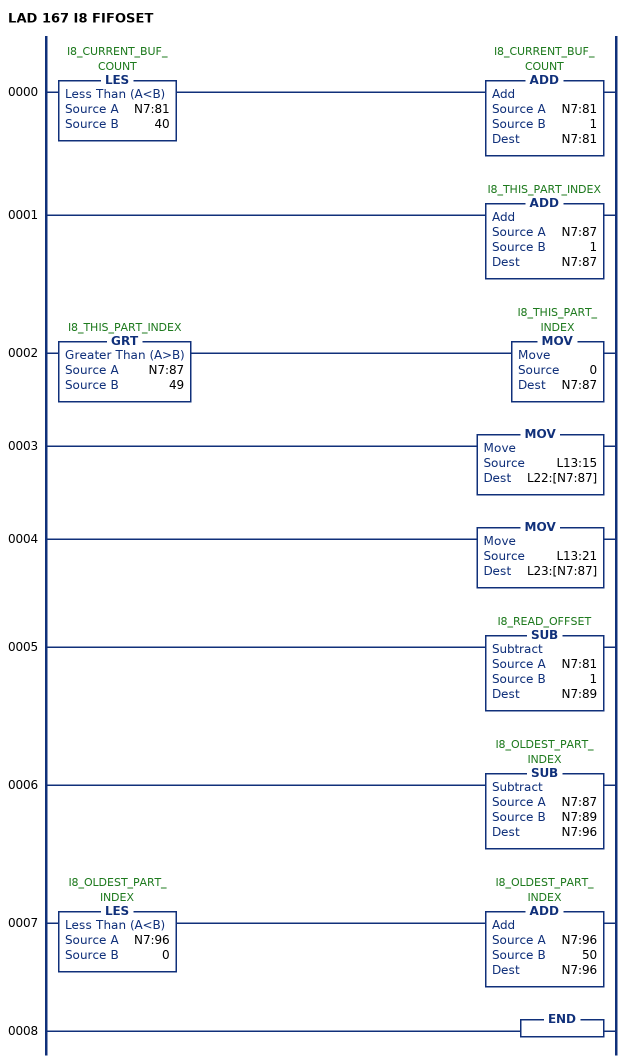
% Rung: 0 %
SOR LES N7:81 40 ADD N7:81 1 N7:81 EOR
%   N7:81  I8_CURRENT_BUF_COUNT %
% Rung: 1 %
SOR ADD N7:87 1 N7:87 EOR
%   N7:87  I8_THIS_PART_INDEX %
% Rung: 2 %
SOR GRT N7:87 49 MOV 0 N7:87 EOR
%   N7:87  I8_THIS_PART_INDEX %
% Rung: 3 %
SOR MOV L13:15 L22:[N7:87] EOR
%   L13:15  THE_TIME %
%   N7:87  I8_THIS_PART_INDEX %
% Rung: 4 %
SOR MOV L13:21 L23:[N7:87] EOR
%   L13:21  TOP_POSITION %
%   N7:87  I8_THIS_PART_INDEX %
% Rung: 5 %
SOR SUB N7:81 1 N7:89 EOR
%   N7:81  I8_CURRENT_BUF_COUNT %
%   N7:89  I8_READ_OFFSET %
% Rung: 6 %
SOR SUB N7:87 N7:89 N7:96 EOR
%   N7:87  I8_THIS_PART_INDEX %
%   N7:89  I8_READ_OFFSET %
%   N7:96  I8_OLDEST_PART_INDEX %
% Rung: 7 %
SOR LES N7:96 0 ADD N7:96 50 N7:96 EOR
%   N7:96  I8_OLDEST_PART_INDEX %
% Rung: 8 %
SOR END EOR

LADDER 168 "I8 FIFOGET"
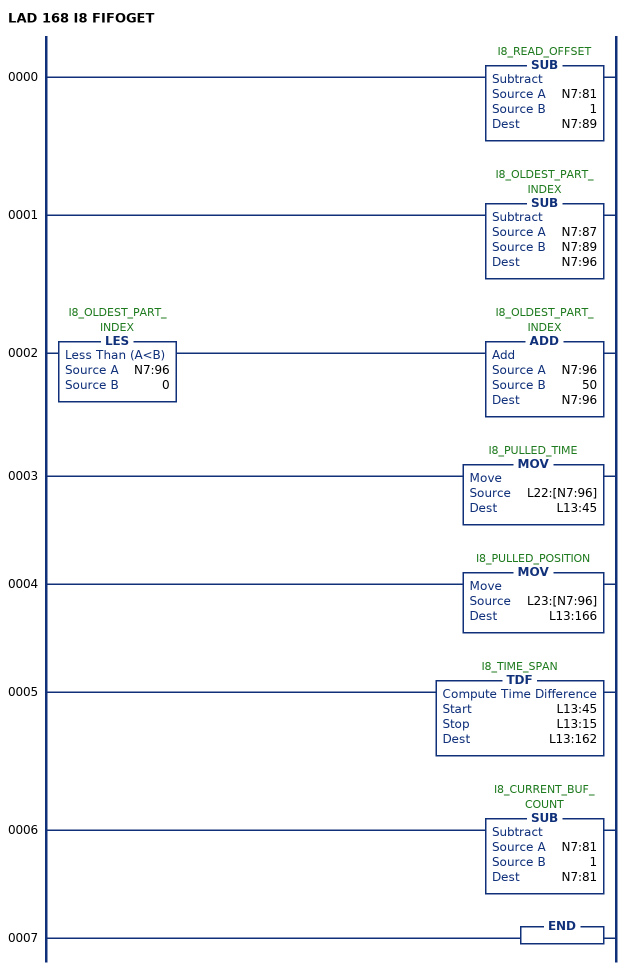
% Rung: 0 %
SOR SUB N7:81 1 N7:89 EOR
%   N7:81  I8_CURRENT_BUF_COUNT %
%   N7:89  I8_READ_OFFSET %
% Rung: 1 %
SOR SUB N7:87 N7:89 N7:96 EOR
%   N7:87  I8_THIS_PART_INDEX %
%   N7:89  I8_READ_OFFSET %
%   N7:96  I8_OLDEST_PART_INDEX %
% Rung: 2 %
SOR LES N7:96 0 ADD N7:96 50 N7:96 EOR
%   N7:96  I8_OLDEST_PART_INDEX %
% Rung: 3 %
SOR MOV L22:[N7:96] L13:45 EOR
%   N7:96  I8_OLDEST_PART_INDEX %
%   L13:45  I8_PULLED_TIME %
% Rung: 4 %
SOR MOV L23:[N7:96] L13:166 EOR
%   N7:96  I8_OLDEST_PART_INDEX %
%   L13:166  I8_PULLED_POSITION %
% Rung: 5 %
SOR TDF L13:45 L13:15 L13:162 EOR
%   L13:45  I8_PULLED_TIME %
%   L13:15  THE_TIME %
%   L13:162  I8_TIME_SPAN %
% Rung: 6 %
SOR SUB N7:81 1 N7:81 EOR
%   N7:81  I8_CURRENT_BUF_COUNT %
% Rung: 7 %
SOR END EOR

LADDER 169 "I8 DATA"
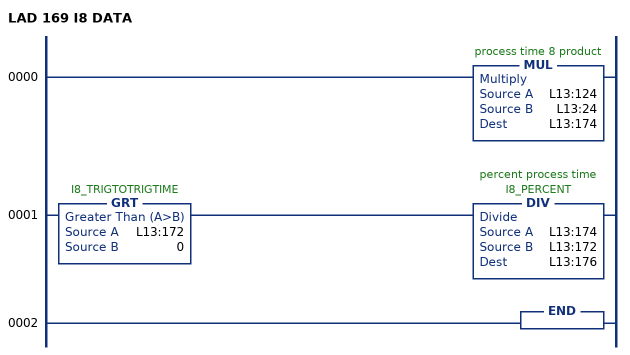
% Rung: 0 %
SOR MUL L13:124 L13:24 L13:174 EOR
%   L13:124  I8_PROCESSTIME %
%   L13:24  "multiplyer to make devision come out to a percentage" %
%   L13:174  "process time 8 product" %
% Rung: 1 %
SOR GRT L13:172 0 DIV L13:174 L13:172 L13:176 EOR
%   L13:172  I8_TRIGTOTRIGTIME %
%   L13:174  "process time 8 product" %
%   L13:176  I8_PERCENT  "percent process time" %
% Rung: 2 %
SOR END EOR

LADDER 170 "I8 FAULT"
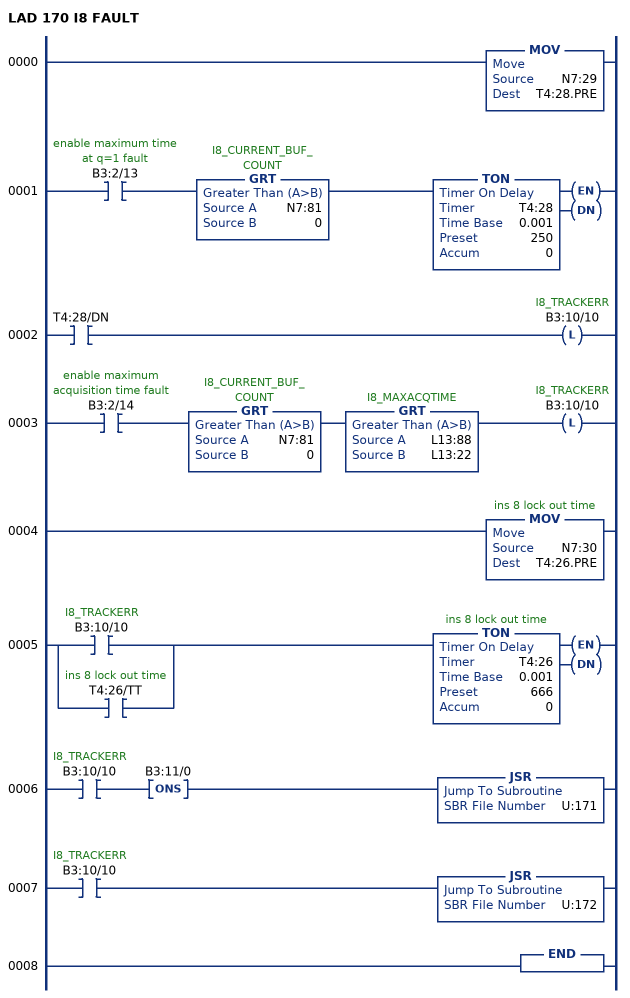
% Rung: 0 %
SOR MOV N7:29 T4:28.PRE EOR
%   N7:29  "max allowed ms time for q to be above 1 if safe fault is used" %
% Rung: 1 %
SOR XIC B3:2/13 GRT N7:81 0 TON T4:28 0.001 250 0 EOR
%   B3:2/13  "enable maximum time at q=1 fault" %
%   N7:81  I8_CURRENT_BUF_COUNT %
% Rung: 2 %
SOR XIC T4:28/DN OTL B3:10/10 EOR
%   B3:10/10  I8_TRACKERR %
% Rung: 3 %
SOR XIC B3:2/14 GRT N7:81 0 GRT L13:88 L13:22 OTL B3:10/10 EOR
%   B3:2/14  "enable maximum acquisition time fault" %
%   N7:81  I8_CURRENT_BUF_COUNT %
%   L13:88  I8_MAXACQTIME %
%   L13:22  "maximum of the longest acquire time allowed if maximum acquire time fault is enabled" %
%   B3:10/10  I8_TRACKERR %
% Rung: 4 %
SOR MOV N7:30 T4:26.PRE EOR
%   N7:30  "ms time setting to lock out inspection to give all pending images a chance to clear" %
%   T4:26  "ins 8 lock out time" %
% Rung: 5 %
SOR BST XIC B3:10/10 NXB XIC T4:26/TT BND TON T4:26 0.001 666 0 EOR
%   B3:10/10  I8_TRACKERR %
%   T4:26  "ins 8 lock out time" %
% Rung: 6 %
SOR XIC B3:10/10 ONS B3:11/0 JSR U:171 EOR
%   B3:10/10  I8_TRACKERR %
% Rung: 7 %
SOR XIC B3:10/10 JSR U:172 EOR
%   B3:10/10  I8_TRACKERR %
% Rung: 8 %
SOR END EOR

LADDER 171 "I8 FIX1"
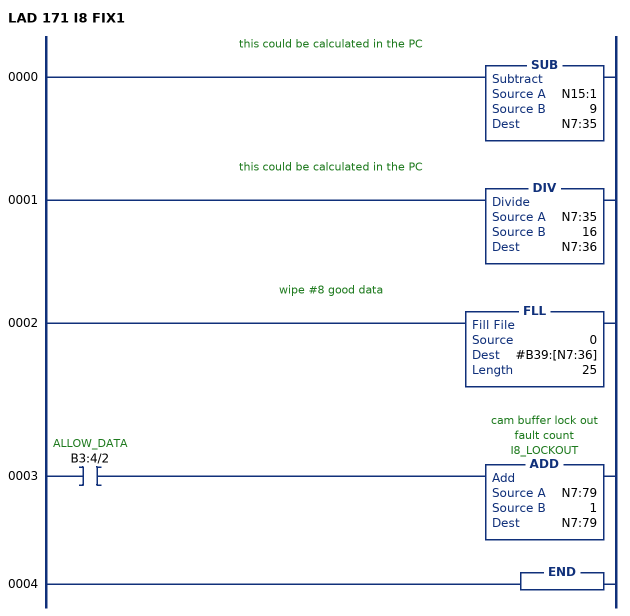
% Rung: 0 %
% this could be calculated in the PC %
SOR SUB N15:1 9 N7:35 EOR
%   N15:1  I8_TRIG_LOC %
% Rung: 1 %
% this could be calculated in the PC %
SOR DIV N7:35 16 N7:36 EOR
% Rung: 2 %
% wipe #8 good data %
SOR FLL 0 #B39:[N7:36] 25 EOR
% Rung: 3 %
SOR XIC B3:4/2 ADD N7:79 1 N7:79 EOR
%   B3:4/2  ALLOW_DATA %
%   N7:79  I8_LOCKOUT  "cam buffer lock out fault count" %
% Rung: 4 %
SOR END EOR

LADDER 172 "I8 FIX2"
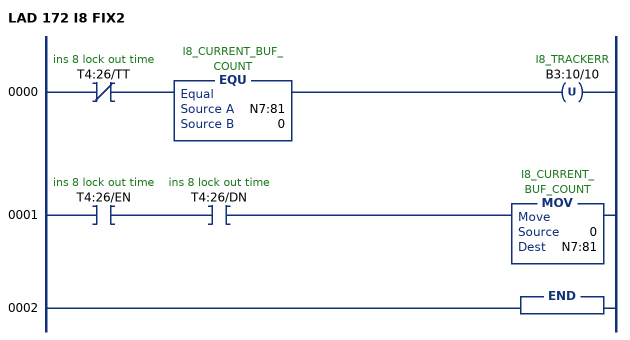
% Rung: 0 %
SOR XIO T4:26/TT EQU N7:81 0 OTU B3:10/10 EOR
%   T4:26  "ins 8 lock out time" %
%   N7:81  I8_CURRENT_BUF_COUNT %
%   B3:10/10  I8_TRACKERR %
% Rung: 1 %
SOR XIC T4:26/EN XIC T4:26/DN MOV 0 N7:81 EOR
%   T4:26  "ins 8 lock out time" %
%   N7:81  I8_CURRENT_BUF_COUNT %
% Rung: 2 %
SOR END EOR

LADDER 200 "PASS BLOW"
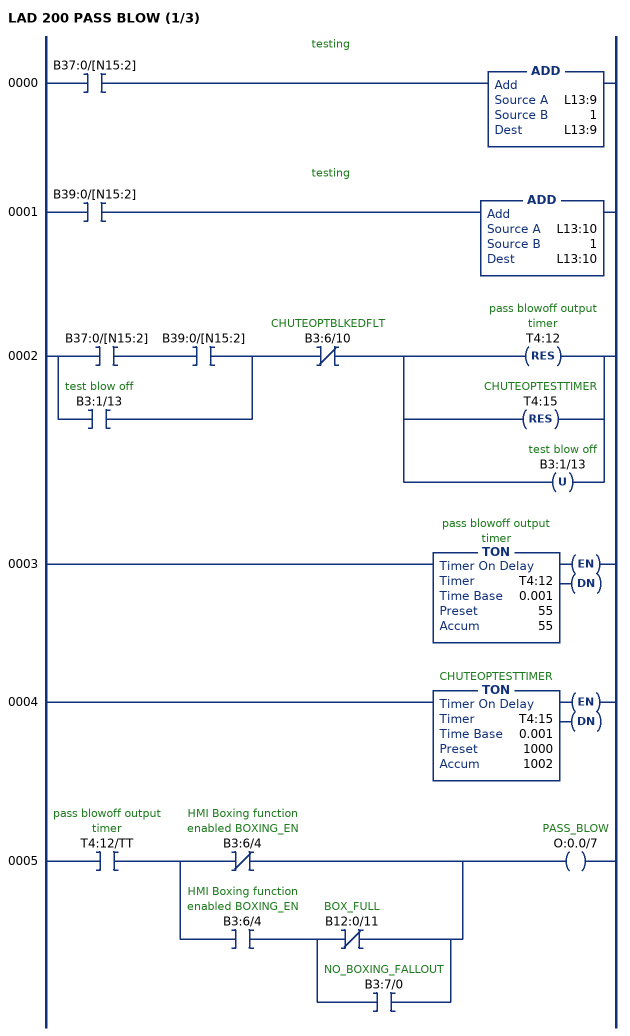
% Rung: 0 %
% testing %
SOR XIC B37:0/[N15:2] ADD L13:9 1 L13:9 EOR
%   B37:0  TOPGOOD1 %
%   N15:2  BLOW_PT %
% Rung: 1 %
% testing %
SOR XIC B39:0/[N15:2] ADD L13:10 1 L13:10 EOR
%   B39:0  TOPGOOD2 %
%   N15:2  BLOW_PT %
% Rung: 2 %
SOR BST XIC B37:0/[N15:2] XIC B39:0/[N15:2] NXB XIC B3:1/13 BND XIO B3:6/10 BST RES T4:12 NXB RES T4:15 NXB OTU B3:1/13 BND EOR
%   B37:0  TOPGOOD1 %
%   N15:2  BLOW_PT %
%   B39:0  TOPGOOD2 %
%   B3:1/13  "test blow off" %
%   B3:6/10  CHUTEOPTBLKEDFLT %
%   T4:12  "pass blowoff output timer" %
%   T4:15  CHUTEOPTESTTIMER %
% Rung: 3 %
SOR TON T4:12 0.001 55 55 EOR
%   T4:12  "pass blowoff output timer" %
% Rung: 4 %
SOR TON T4:15 0.001 1000 1002 EOR
%   T4:15  CHUTEOPTESTTIMER %
% Rung: 5 %
SOR XIC T4:12/TT BST XIO B3:6/4 NXB XIC B3:6/4 BST XIO B12:0/11 NXB XIC B3:7/0 BND BND OTE O:0.0/7 EOR
%   T4:12  "pass blowoff output timer" %
%   B3:6/4  BOXING_EN  "HMI Boxing function enabled" %
%   B12:0/11  BOX_FULL %
%   B3:7/0  NO_BOXING_FALLOUT %
%   O:0.0/7  PASS_BLOW %

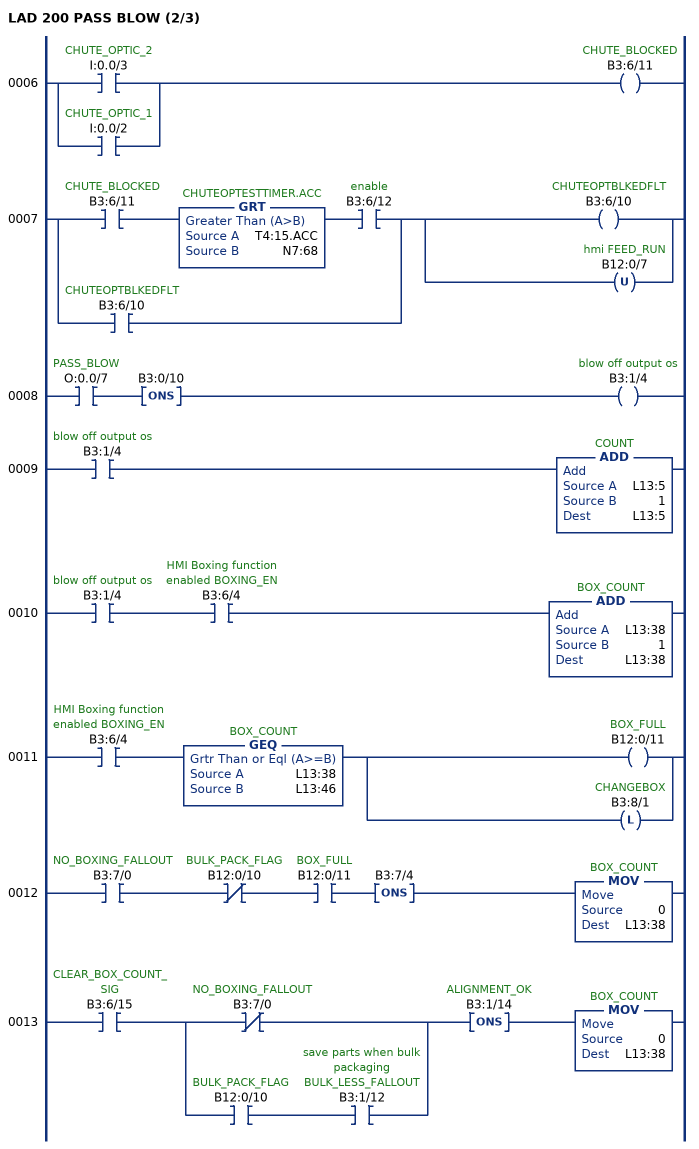
% Rung: 6 %
SOR BST XIC I:0.0/3 NXB XIC I:0.0/2 BND OTE B3:6/11 EOR
%   I:0.0/3  CHUTE_OPTIC_2 %
%   I:0.0/2  CHUTE_OPTIC_1 %
%   B3:6/11  CHUTE_BLOCKED %
% Rung: 7 %
SOR BST XIC B3:6/11 GRT T4:15.ACC N7:68 XIC B3:6/12 NXB XIC B3:6/10 BND BST OTE B3:6/10 NXB OTU B12:0/7 BND EOR
%   B3:6/11  CHUTE_BLOCKED %
%   T4:15  CHUTEOPTESTTIMER %
%   B3:6/12  "enable" %
%   B3:6/10  CHUTEOPTBLKEDFLT %
%   B12:0/7  FEED_RUN  "hmi" %
% Rung: 8 %
SOR XIC O:0.0/7 ONS B3:0/10 OTE B3:1/4 EOR
%   O:0.0/7  PASS_BLOW %
%   B3:1/4  "blow off output os" %
% Rung: 9 %
SOR XIC B3:1/4 ADD L13:5 1 L13:5 EOR
%   B3:1/4  "blow off output os" %
%   L13:5  COUNT %
% Rung: 10 %
SOR XIC B3:1/4 XIC B3:6/4 ADD L13:38 1 L13:38 EOR
%   B3:1/4  "blow off output os" %
%   B3:6/4  BOXING_EN  "HMI Boxing function enabled" %
%   L13:38  BOX_COUNT %
% Rung: 11 %
SOR XIC B3:6/4 GEQ L13:38 L13:46 BST OTE B12:0/11 NXB OTL B3:8/1 BND EOR
%   B3:6/4  BOXING_EN  "HMI Boxing function enabled" %
%   L13:38  BOX_COUNT %
%   L13:46  BOX_LIMIT  "box count setpoint" %
%   B12:0/11  BOX_FULL %
%   B3:8/1  CHANGEBOX %
% Rung: 12 %
SOR XIC B3:7/0 XIO B12:0/10 XIC B12:0/11 ONS B3:7/4 MOV 0 L13:38 EOR
%   B3:7/0  NO_BOXING_FALLOUT %
%   B12:0/10  BULK_PACK_FLAG %
%   B12:0/11  BOX_FULL %
%   L13:38  BOX_COUNT %
% Rung: 13 %
SOR XIC B3:6/15 BST XIO B3:7/0 NXB XIC B12:0/10 XIC B3:1/12 BND ONS B3:1/14 MOV 0 L13:38 EOR
%   B3:6/15  CLEAR_BOX_COUNT_SIG %
%   B3:7/0  NO_BOXING_FALLOUT %
%   B12:0/10  BULK_PACK_FLAG %
%   B3:1/12  BULK_LESS_FALLOUT  "save parts when bulk packaging" %
%   B3:1/14  ALIGNMENT_OK %
%   L13:38  BOX_COUNT %

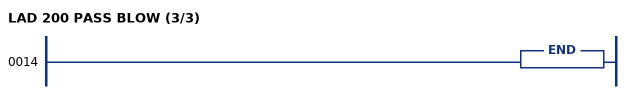
% Rung: 14 %
SOR END EOR

LADDER 213 "TESTTRIG1"
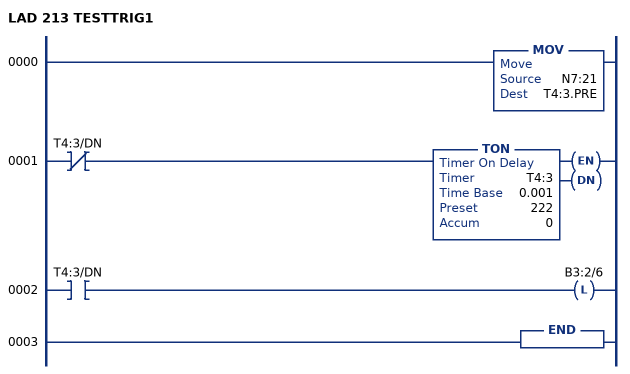
% Rung: 0 %
SOR MOV N7:21 T4:3.PRE EOR
% Rung: 1 %
SOR XIO T4:3/DN TON T4:3 0.001 222 0 EOR
% Rung: 2 %
SOR XIC T4:3/DN OTL B3:2/6 EOR
% Rung: 3 %
SOR END EOR

LADDER 214 "TESTTRIG5"
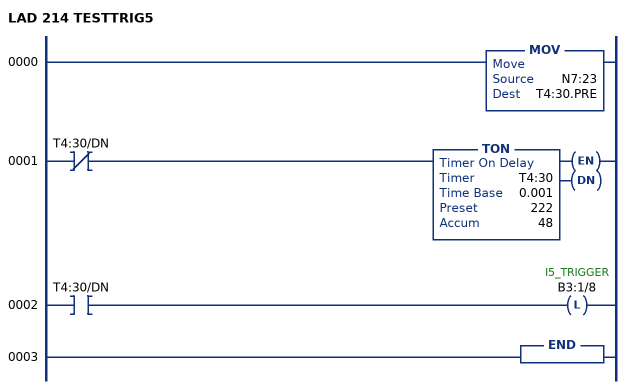
% Rung: 0 %
SOR MOV N7:23 T4:30.PRE EOR
%   N7:23  I5_TRIGTIME %
% Rung: 1 %
SOR XIO T4:30/DN TON T4:30 0.001 222 48 EOR
% Rung: 2 %
SOR XIC T4:30/DN OTL B3:1/8 EOR
%   B3:1/8  I5_TRIGGER %
% Rung: 3 %
SOR END EOR

LADDER 215 "TESTTRIG6"
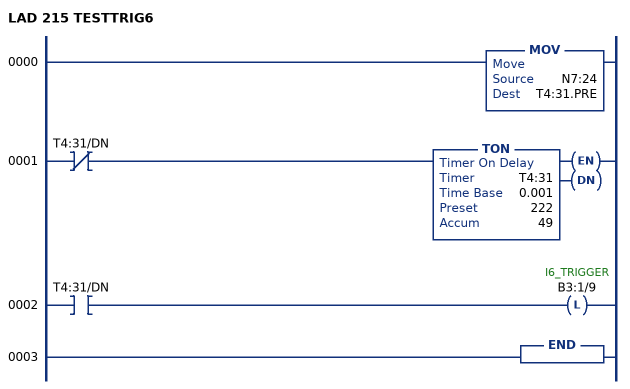
% Rung: 0 %
SOR MOV N7:24 T4:31.PRE EOR
%   N7:24  I6_TRIGTIME %
% Rung: 1 %
SOR XIO T4:31/DN TON T4:31 0.001 222 49 EOR
% Rung: 2 %
SOR XIC T4:31/DN OTL B3:1/9 EOR
%   B3:1/9  I6_TRIGGER %
% Rung: 3 %
SOR END EOR

LADDER 216 "TESTTRIG7"
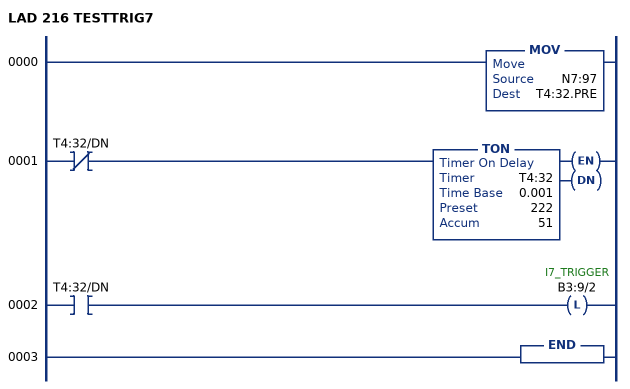
% Rung: 0 %
SOR MOV N7:97 T4:32.PRE EOR
%   N7:97  I7_TRIGTIME %
% Rung: 1 %
SOR XIO T4:32/DN TON T4:32 0.001 222 51 EOR
% Rung: 2 %
SOR XIC T4:32/DN OTL B3:9/2 EOR
%   B3:9/2  I7_TRIGGER %
% Rung: 3 %
SOR END EOR

LADDER 217 "TESTTRIG8"
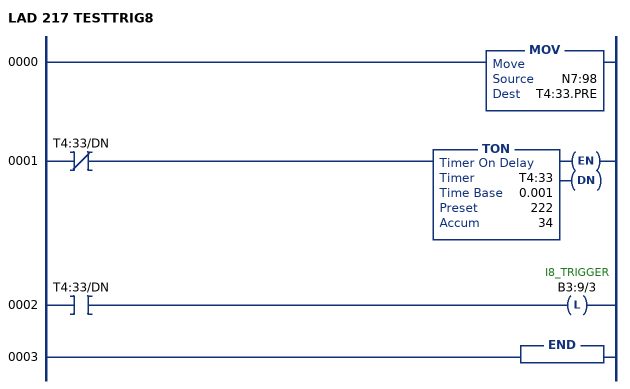
% Rung: 0 %
SOR MOV N7:98 T4:33.PRE EOR
%   N7:98  I8_TRIGTIME %
% Rung: 1 %
SOR XIO T4:33/DN TON T4:33 0.001 222 34 EOR
% Rung: 2 %
SOR XIC T4:33/DN OTL B3:9/3 EOR
%   B3:9/3  I8_TRIGGER %
% Rung: 3 %
SOR END EOR

LADDER 219 "PACKAGER"    % normal %
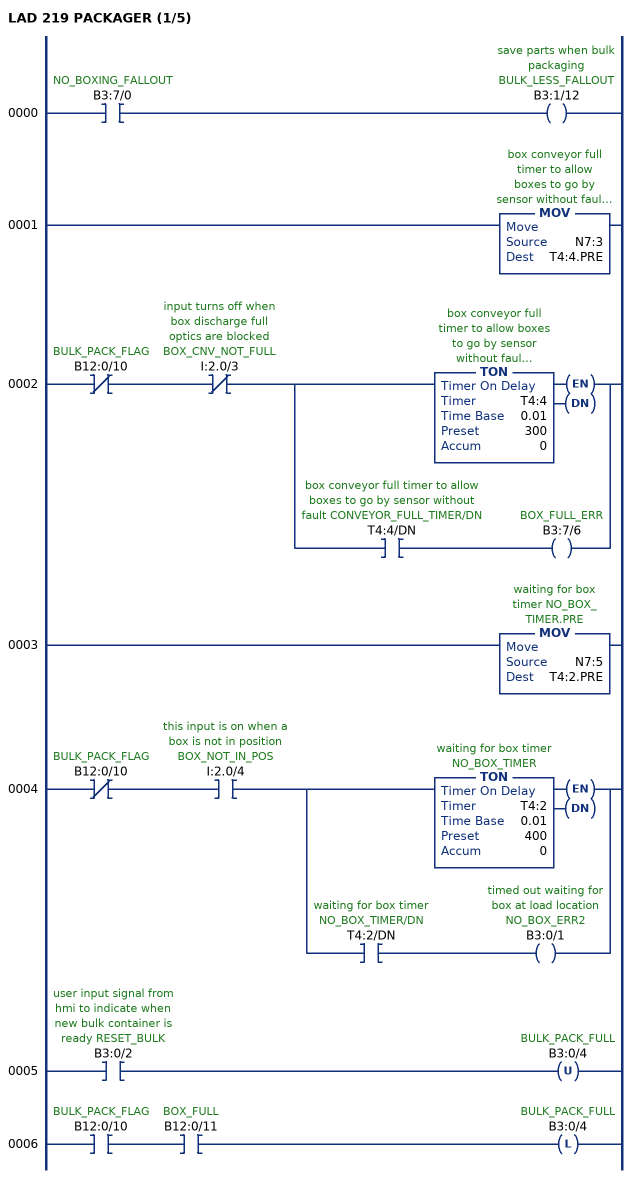
% Rung: 0 %
SOR XIC B3:7/0 OTE B3:1/12 EOR
%   B3:7/0  NO_BOXING_FALLOUT %
%   B3:1/12  BULK_LESS_FALLOUT  "save parts when bulk packaging" %
% Rung: 1 %
SOR MOV N7:3 T4:4.PRE EOR
%   N7:3  "time to allow box to pass box conveyor full sensor without fault" %
%   T4:4  CONVEYOR_FULL_TIMER  "box conveyor full timer to allow boxes to go by sensor without fault" %
% Rung: 2 %
SOR XIO B12:0/10 XIO I:2.0/3 BST TON T4:4 0.01 300 0 NXB XIC T4:4/DN OTE B3:7/6 BND EOR
%   B12:0/10  BULK_PACK_FLAG %
%   I:2.0/3  BOX_CNV_NOT_FULL  "input turns off when box discharge full optics are blocked" %
%   T4:4  CONVEYOR_FULL_TIMER  "box conveyor full timer to allow boxes to go by sensor without fault" %
%   B3:7/6  BOX_FULL_ERR %
% Rung: 3 %
SOR MOV N7:5 T4:2.PRE EOR
%   N7:5  "buffer count 6" %
%   T4:2  NO_BOX_TIMER  "waiting for box timer" %
% Rung: 4 %
SOR XIO B12:0/10 XIC I:2.0/4 BST TON T4:2 0.01 400 0 NXB XIC T4:2/DN OTE B3:0/1 BND EOR
%   B12:0/10  BULK_PACK_FLAG %
%   I:2.0/4  BOX_NOT_IN_POS  "this input is on when a box is not in position" %
%   T4:2  NO_BOX_TIMER  "waiting for box timer" %
%   B3:0/1  NO_BOX_ERR2  "timed out waiting for box at load location" %
% Rung: 5 %
SOR XIC B3:0/2 OTU B3:0/4 EOR
%   B3:0/2  RESET_BULK  "user input signal from hmi to indicate when new bulk container is ready" %
%   B3:0/4  BULK_PACK_FULL %
% Rung: 6 %
SOR XIC B12:0/10 XIC B12:0/11 OTL B3:0/4 EOR
%   B12:0/10  BULK_PACK_FLAG %
%   B12:0/11  BOX_FULL %
%   B3:0/4  BULK_PACK_FULL %

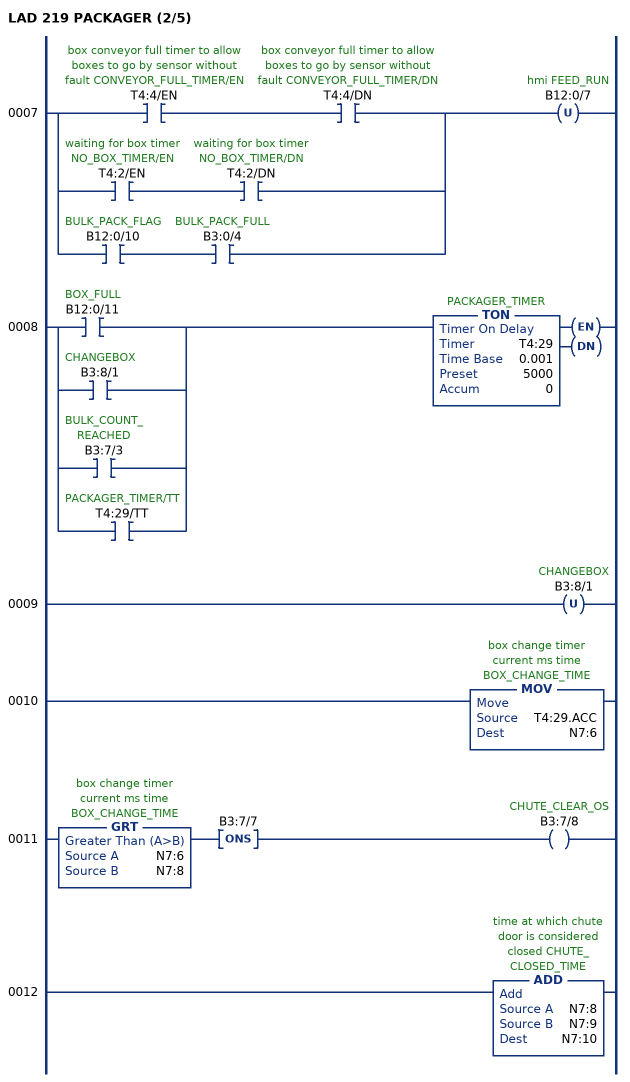
% Rung: 7 %
SOR BST XIC T4:4/EN XIC T4:4/DN NXB XIC T4:2/EN XIC T4:2/DN NXB XIC B12:0/10 XIC B3:0/4 BND OTU B12:0/7 EOR
%   T4:4  CONVEYOR_FULL_TIMER  "box conveyor full timer to allow boxes to go by sensor without fault" %
%   T4:2  NO_BOX_TIMER  "waiting for box timer" %
%   B12:0/10  BULK_PACK_FLAG %
%   B3:0/4  BULK_PACK_FULL %
%   B12:0/7  FEED_RUN  "hmi" %
% Rung: 8 %
SOR BST XIC B12:0/11 NXB XIC B3:8/1 NXB XIC B3:7/3 NXB XIC T4:29/TT BND TON T4:29 0.001 5000 0 EOR
%   B12:0/11  BOX_FULL %
%   B3:8/1  CHANGEBOX %
%   B3:7/3  BULK_COUNT_REACHED %
%   T4:29  PACKAGER_TIMER %
% Rung: 9 %
SOR OTU B3:8/1 EOR
%   B3:8/1  CHANGEBOX %
% Rung: 10 %
SOR MOV T4:29.ACC N7:6 EOR
%   T4:29  PACKAGER_TIMER %
%   N7:6  BOX_CHANGE_TIME  "box change timer current ms time" %
% Rung: 11 %
SOR GRT N7:6 N7:8 ONS B3:7/7 OTE B3:7/8 EOR
%   N7:6  BOX_CHANGE_TIME  "box change timer current ms time" %
%   N7:8  CHUTE_CLEAR_TIME %
%   B3:7/8  CHUTE_CLEAR_OS %
% Rung: 12 %
SOR ADD N7:8 N7:9 N7:10 EOR
%   N7:8  CHUTE_CLEAR_TIME %
%   N7:9  CHUTE_CLOSE_TIME  "ms time required to close chute" %
%   N7:10  CHUTE_CLOSED_TIME  "time at which chute door is considered closed" %

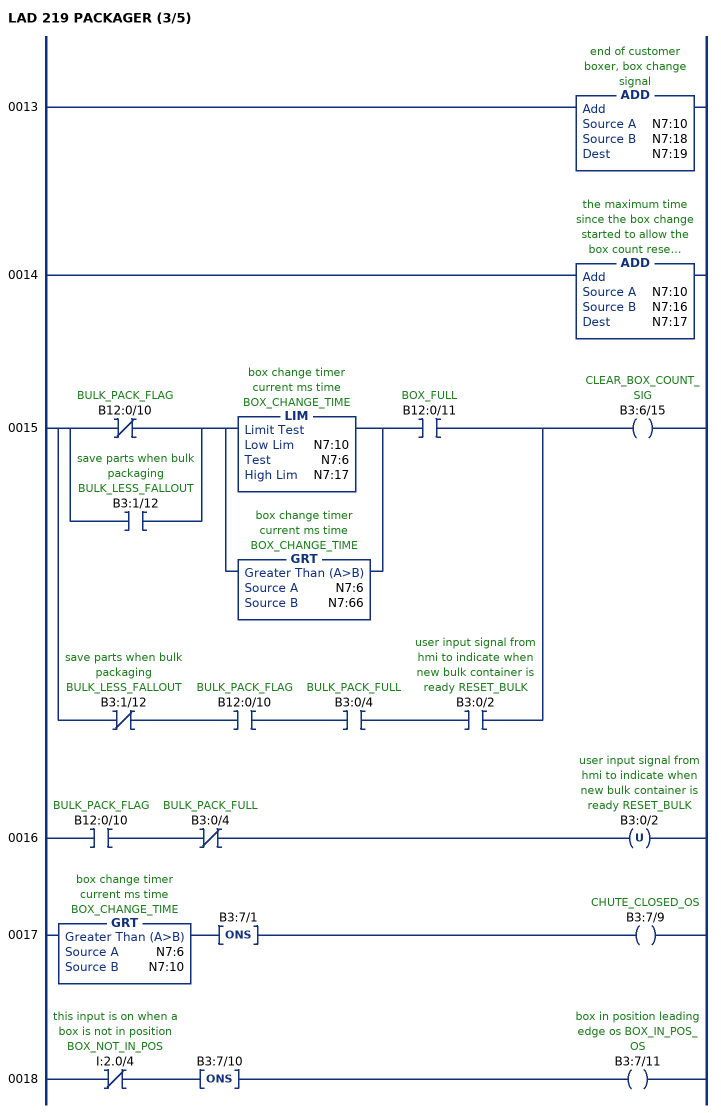
% Rung: 13 %
SOR ADD N7:10 N7:18 N7:19 EOR
%   N7:10  CHUTE_CLOSED_TIME  "time at which chute door is considered closed" %
%   N7:18  CHANGE_BOX_SIG_TIME  "customer boxer change box signal time" %
%   N7:19  "end of customer boxer, box change signal" %
% Rung: 14 %
SOR ADD N7:10 N7:16 N7:17 EOR
%   N7:10  CHUTE_CLOSED_TIME  "time at which chute door is considered closed" %
%   N7:16  RESET_COUNT_SIG_TIME  "maximum length of time to hold box count reset signal on" %
%   N7:17  "the maximum time since the box change started to allow the box count reset signal" %
% Rung: 15 %
SOR BST BST XIO B12:0/10 NXB XIC B3:1/12 BND BST LIM N7:10 N7:6 N7:17 NXB GRT N7:6 N7:66 BND XIC B12:0/11 NXB XIO B3:1/12 XIC B12:0/10 XIC B3:0/4 XIC B3:0/2 BND OTE B3:6/15 EOR
%   B12:0/10  BULK_PACK_FLAG %
%   B3:1/12  BULK_LESS_FALLOUT  "save parts when bulk packaging" %
%   N7:10  CHUTE_CLOSED_TIME  "time at which chute door is considered closed" %
%   N7:6  BOX_CHANGE_TIME  "box change timer current ms time" %
%   N7:17  "the maximum time since the box change started to allow the box count reset signal" %
%   B12:0/11  BOX_FULL %
%   B3:0/4  BULK_PACK_FULL %
%   B3:0/2  RESET_BULK  "user input signal from hmi to indicate when new bulk container is ready" %
%   B3:6/15  CLEAR_BOX_COUNT_SIG %
% Rung: 16 %
SOR XIC B12:0/10 XIO B3:0/4 OTU B3:0/2 EOR
%   B12:0/10  BULK_PACK_FLAG %
%   B3:0/4  BULK_PACK_FULL %
%   B3:0/2  RESET_BULK  "user input signal from hmi to indicate when new bulk container is ready" %
% Rung: 17 %
SOR GRT N7:6 N7:10 ONS B3:7/1 OTE B3:7/9 EOR
%   N7:6  BOX_CHANGE_TIME  "box change timer current ms time" %
%   N7:10  CHUTE_CLOSED_TIME  "time at which chute door is considered closed" %
%   B3:7/9  CHUTE_CLOSED_OS %
% Rung: 18 %
SOR XIO I:2.0/4 ONS B3:7/10 OTE B3:7/11 EOR
%   I:2.0/4  BOX_NOT_IN_POS  "this input is on when a box is not in position" %
%   B3:7/11  BOX_IN_POS_OS  "box in position leading edge os" %

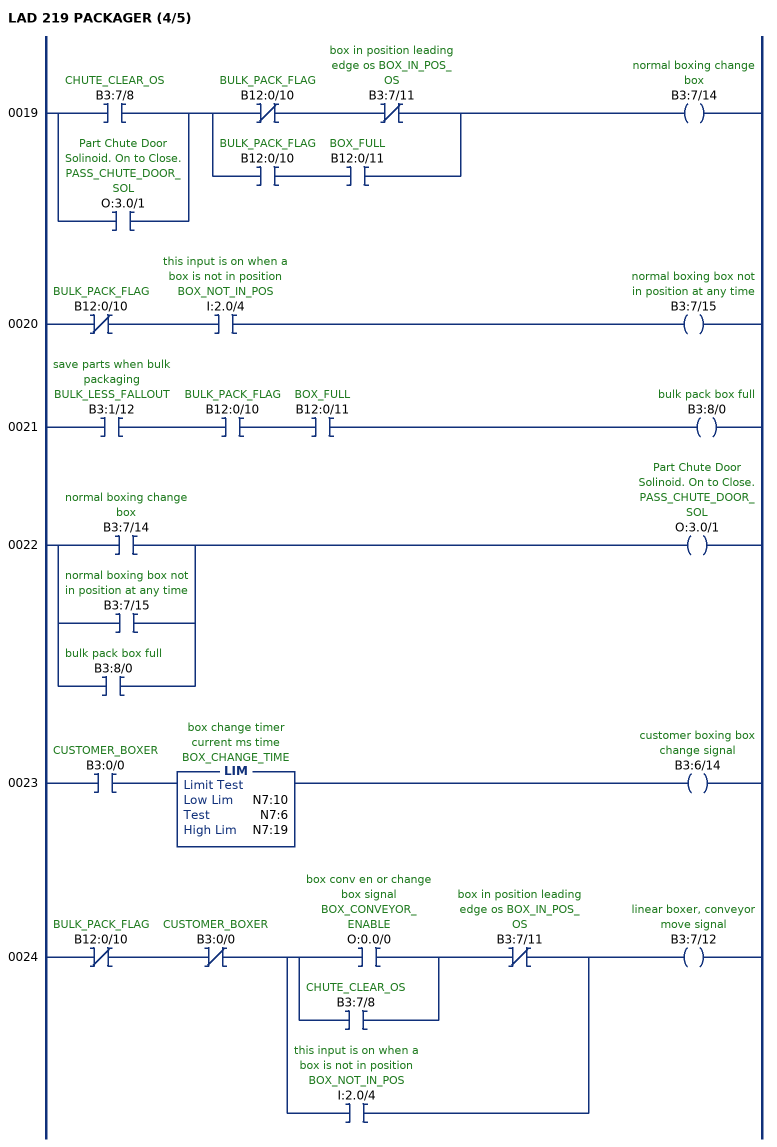
% Rung: 19 %
SOR BST XIC B3:7/8 NXB XIC O:3.0/1 BND BST XIO B12:0/10 XIO B3:7/11 NXB XIC B12:0/10 XIC B12:0/11 BND OTE B3:7/14 EOR
%   B3:7/8  CHUTE_CLEAR_OS %
%   O:3.0/1  PASS_CHUTE_DOOR_SOL  "Part Chute Door Solinoid. On to Close." %
%   B12:0/10  BULK_PACK_FLAG %
%   B3:7/11  BOX_IN_POS_OS  "box in position leading edge os" %
%   B12:0/11  BOX_FULL %
%   B3:7/14  "normal boxing change box" %
% Rung: 20 %
SOR XIO B12:0/10 XIC I:2.0/4 OTE B3:7/15 EOR
%   B12:0/10  BULK_PACK_FLAG %
%   I:2.0/4  BOX_NOT_IN_POS  "this input is on when a box is not in position" %
%   B3:7/15  "normal boxing box not in position at any time" %
% Rung: 21 %
SOR XIC B3:1/12 XIC B12:0/10 XIC B12:0/11 OTE B3:8/0 EOR
%   B3:1/12  BULK_LESS_FALLOUT  "save parts when bulk packaging" %
%   B12:0/10  BULK_PACK_FLAG %
%   B12:0/11  BOX_FULL %
%   B3:8/0  "bulk pack box full" %
% Rung: 22 %
SOR BST XIC B3:7/14 NXB XIC B3:7/15 NXB XIC B3:8/0 BND OTE O:3.0/1 EOR
%   B3:7/14  "normal boxing change box" %
%   B3:7/15  "normal boxing box not in position at any time" %
%   B3:8/0  "bulk pack box full" %
%   O:3.0/1  PASS_CHUTE_DOOR_SOL  "Part Chute Door Solinoid. On to Close." %
% Rung: 23 %
SOR XIC B3:0/0 LIM N7:10 N7:6 N7:19 OTE B3:6/14 EOR
%   B3:0/0  CUSTOMER_BOXER %
%   N7:10  CHUTE_CLOSED_TIME  "time at which chute door is considered closed" %
%   N7:6  BOX_CHANGE_TIME  "box change timer current ms time" %
%   N7:19  "end of customer boxer, box change signal" %
%   B3:6/14  "customer boxing box change signal" %
% Rung: 24 %
SOR XIO B12:0/10 XIO B3:0/0 BST BST XIC O:0.0/0 NXB XIC B3:7/8 BND XIO B3:7/11 NXB XIC I:2.0/4 BND OTE B3:7/12 EOR
%   B12:0/10  BULK_PACK_FLAG %
%   B3:0/0  CUSTOMER_BOXER %
%   O:0.0/0  BOX_CONVEYOR_ENABLE  "box conv en or change box signal" %
%   B3:7/8  CHUTE_CLEAR_OS %
%   B3:7/11  BOX_IN_POS_OS  "box in position leading edge os" %
%   I:2.0/4  BOX_NOT_IN_POS  "this input is on when a box is not in position" %
%   B3:7/12  "linear boxer, conveyor move signal" %

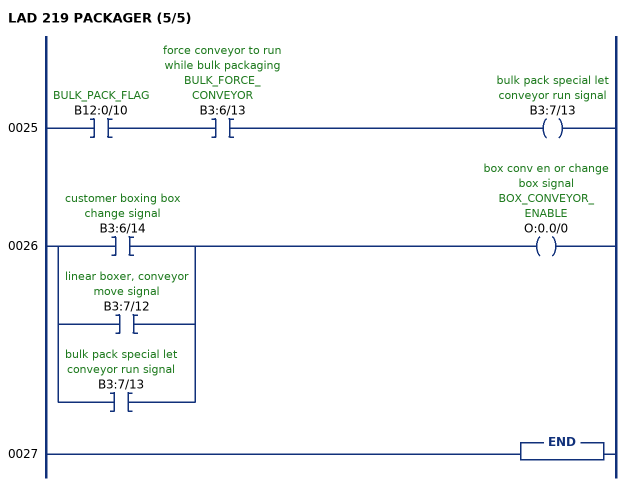
% Rung: 25 %
SOR XIC B12:0/10 XIC B3:6/13 OTE B3:7/13 EOR
%   B12:0/10  BULK_PACK_FLAG %
%   B3:6/13  BULK_FORCE_CONVEYOR  "force conveyor to run while bulk packaging" %
%   B3:7/13  "bulk pack special let conveyor run signal" %
% Rung: 26 %
SOR BST XIC B3:6/14 NXB XIC B3:7/12 NXB XIC B3:7/13 BND OTE O:0.0/0 EOR
%   B3:6/14  "customer boxing box change signal" %
%   B3:7/12  "linear boxer, conveyor move signal" %
%   B3:7/13  "bulk pack special let conveyor run signal" %
%   O:0.0/0  BOX_CONVEYOR_ENABLE  "box conv en or change box signal" %
% Rung: 27 %
SOR END EOR

LADDER 220 "NO PACKAGE"
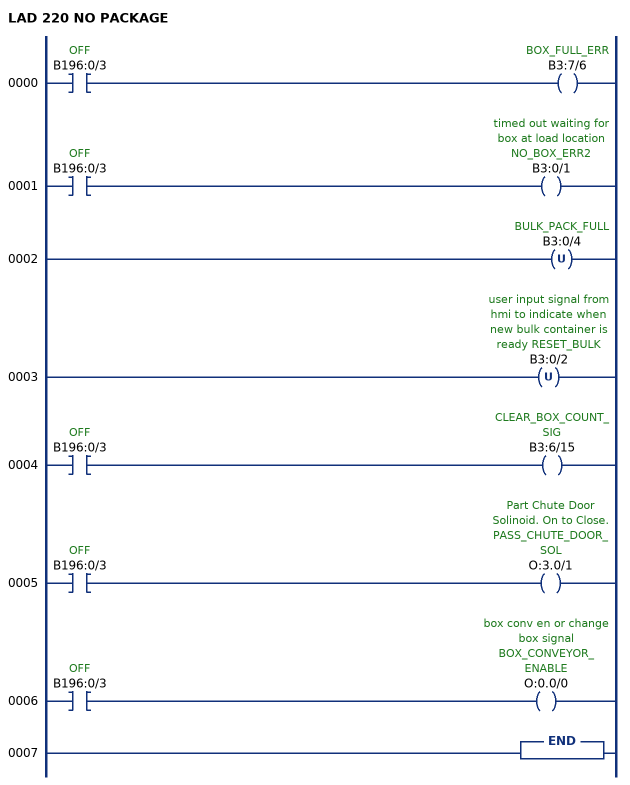
% Rung: 0 %
SOR XIC B196:0/3 OTE B3:7/6 EOR
%   B196:0/3  OFF %
%   B3:7/6  BOX_FULL_ERR %
% Rung: 1 %
SOR XIC B196:0/3 OTE B3:0/1 EOR
%   B196:0/3  OFF %
%   B3:0/1  NO_BOX_ERR2  "timed out waiting for box at load location" %
% Rung: 2 %
SOR OTU B3:0/4 EOR
%   B3:0/4  BULK_PACK_FULL %
% Rung: 3 %
SOR OTU B3:0/2 EOR
%   B3:0/2  RESET_BULK  "user input signal from hmi to indicate when new bulk container is ready" %
% Rung: 4 %
SOR XIC B196:0/3 OTE B3:6/15 EOR
%   B196:0/3  OFF %
%   B3:6/15  CLEAR_BOX_COUNT_SIG %
% Rung: 5 %
SOR XIC B196:0/3 OTE O:3.0/1 EOR
%   B196:0/3  OFF %
%   O:3.0/1  PASS_CHUTE_DOOR_SOL  "Part Chute Door Solinoid. On to Close." %
% Rung: 6 %
SOR XIC B196:0/3 OTE O:0.0/0 EOR
%   B196:0/3  OFF %
%   O:0.0/0  BOX_CONVEYOR_ENABLE  "box conv en or change box signal" %
% Rung: 7 %
SOR END EOR

LADDER 222 "RATE1"
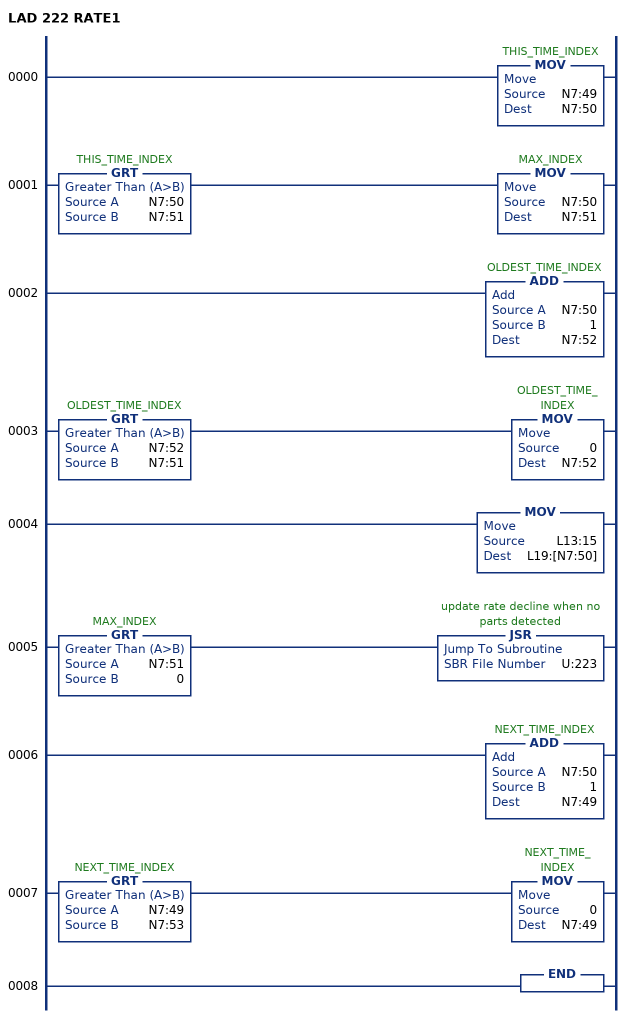
% Rung: 0 %
SOR MOV N7:49 N7:50 EOR
%   N7:49  NEXT_TIME_INDEX %
%   N7:50  THIS_TIME_INDEX %
% Rung: 1 %
SOR GRT N7:50 N7:51 MOV N7:50 N7:51 EOR
%   N7:50  THIS_TIME_INDEX %
%   N7:51  MAX_INDEX %
% Rung: 2 %
SOR ADD N7:50 1 N7:52 EOR
%   N7:50  THIS_TIME_INDEX %
%   N7:52  OLDEST_TIME_INDEX %
% Rung: 3 %
SOR GRT N7:52 N7:51 MOV 0 N7:52 EOR
%   N7:52  OLDEST_TIME_INDEX %
%   N7:51  MAX_INDEX %
% Rung: 4 %
SOR MOV L13:15 L19:[N7:50] EOR
%   L13:15  THE_TIME %
%   N7:50  THIS_TIME_INDEX %
% Rung: 5 %
SOR GRT N7:51 0 JSR U:223 EOR
%   N7:51  MAX_INDEX %
%   U:223  "update rate decline when no parts detected" %
% Rung: 6 %
SOR ADD N7:50 1 N7:49 EOR
%   N7:50  THIS_TIME_INDEX %
%   N7:49  NEXT_TIME_INDEX %
% Rung: 7 %
SOR GRT N7:49 N7:53 MOV 0 N7:49 EOR
%   N7:49  NEXT_TIME_INDEX %
%   N7:53  UPPER_INDEX_LIMIT %
% Rung: 8 %
SOR END EOR

LADDER 223 "RATE2"
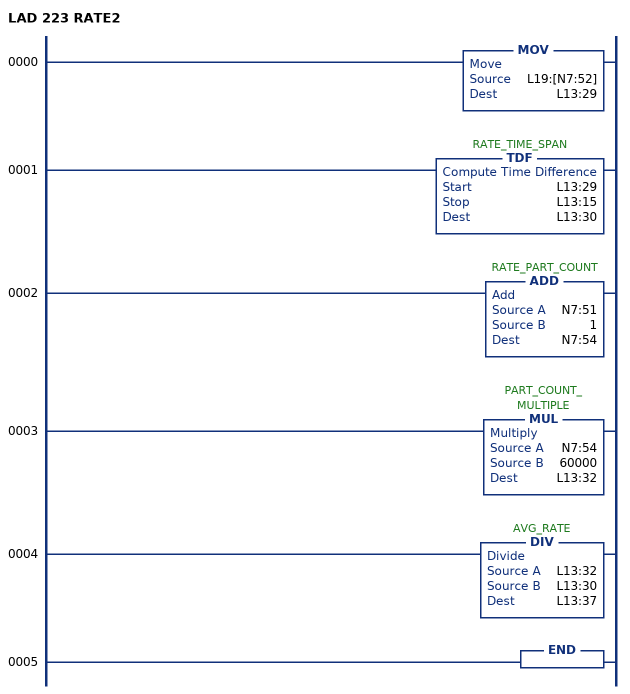
% Rung: 0 %
SOR MOV L19:[N7:52] L13:29 EOR
%   N7:52  OLDEST_TIME_INDEX %
% Rung: 1 %
SOR TDF L13:29 L13:15 L13:30 EOR
%   L13:15  THE_TIME %
%   L13:30  RATE_TIME_SPAN %
% Rung: 2 %
SOR ADD N7:51 1 N7:54 EOR
%   N7:51  MAX_INDEX %
%   N7:54  RATE_PART_COUNT %
% Rung: 3 %
SOR MUL N7:54 60000 L13:32 EOR
%   N7:54  RATE_PART_COUNT %
%   L13:32  PART_COUNT_MULTIPLE %
% Rung: 4 %
SOR DIV L13:32 L13:30 L13:37 EOR
%   L13:32  PART_COUNT_MULTIPLE %
%   L13:30  RATE_TIME_SPAN %
%   L13:37  AVG_RATE %
% Rung: 5 %
SOR END EOR

LADDER 224 "RESET RATE"
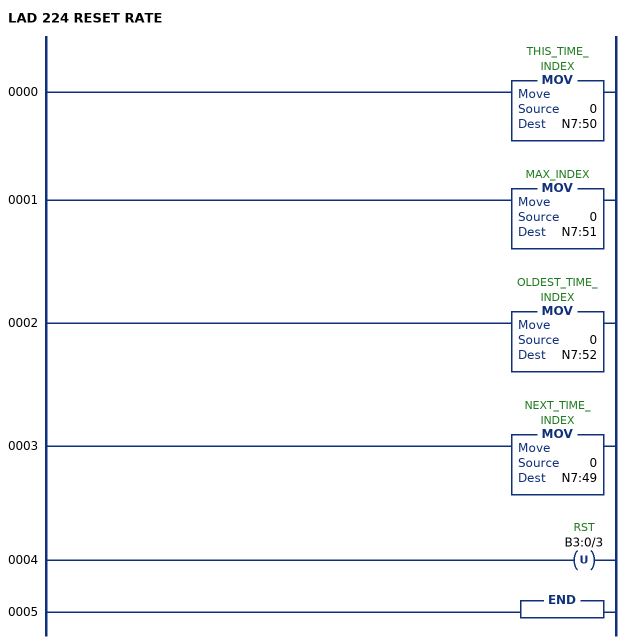
% Rung: 0 %
SOR MOV 0 N7:50 EOR
%   N7:50  THIS_TIME_INDEX %
% Rung: 1 %
SOR MOV 0 N7:51 EOR
%   N7:51  MAX_INDEX %
% Rung: 2 %
SOR MOV 0 N7:52 EOR
%   N7:52  OLDEST_TIME_INDEX %
% Rung: 3 %
SOR MOV 0 N7:49 EOR
%   N7:49  NEXT_TIME_INDEX %
% Rung: 4 %
SOR OTU B3:0/3 EOR
%   B3:0/3  RST %
% Rung: 5 %
SOR END EOR

LADDER 240 "NP STOP"
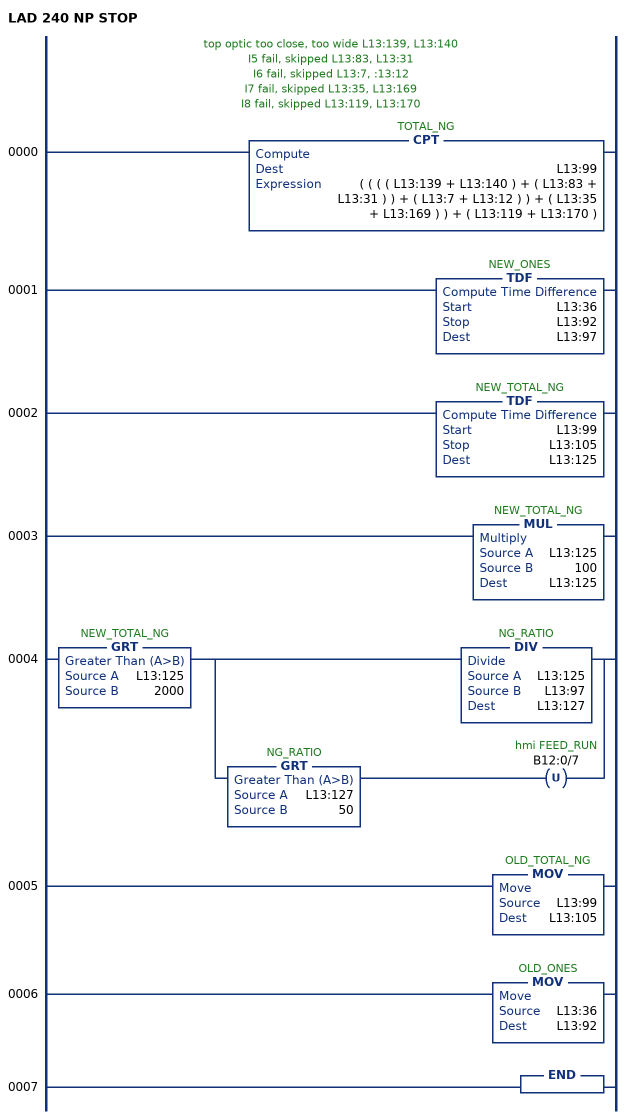
% Rung: 0 %
% top optic too close, too wide L13:139, L13:140
% I5 fail, skipped L13:83, L13:31
% I6 fail, skipped L13:7, :13:12
% I7 fail, skipped L13:35, L13:169
% I8 fail, skipped L13:119, L13:170 %
SOR CPT L13:99 " ( ( ( ( L13:139 + L13:140 ) + ( L13:83 + L13:31 ) ) + ( L13:7 + L13:12 ) ) + ( L13:35 + L13:169 ) ) + ( L13:119 + L13:170 ) " EOR
%   L13:99  TOTAL_NG %
%   L13:139  "too close top count" %
%   L13:140  "too wide top count" %
%   L13:83  I5_FAIL_COUNT %
%   L13:31  I5_SKIPPEDCOUNT %
%   L13:7  I6_FAIL_COUNT %
%   L13:12  I6_SKIPPEDCOUNT %
%   L13:35  I7_FAIL_COUNT %
%   L13:169  I7_SKIPPEDCOUNT %
%   L13:119  I8_FAIL_COUNT %
%   L13:170  I8_SKIPPEDCOUNT %
% Rung: 1 %
SOR TDF L13:36 L13:92 L13:97 EOR
%   L13:36  ONES %
%   L13:92  OLD_ONES %
%   L13:97  NEW_ONES %
% Rung: 2 %
SOR TDF L13:99 L13:105 L13:125 EOR
%   L13:99  TOTAL_NG %
%   L13:105  OLD_TOTAL_NG %
%   L13:125  NEW_TOTAL_NG %
% Rung: 3 %
SOR MUL L13:125 100 L13:125 EOR
%   L13:125  NEW_TOTAL_NG %
% Rung: 4 %
SOR GRT L13:125 2000 BST DIV L13:125 L13:97 L13:127 NXB GRT L13:127 50 OTU B12:0/7 BND EOR
%   L13:125  NEW_TOTAL_NG %
%   L13:97  NEW_ONES %
%   L13:127  NG_RATIO %
%   B12:0/7  FEED_RUN  "hmi" %
% Rung: 5 %
SOR MOV L13:99 L13:105 EOR
%   L13:99  TOTAL_NG %
%   L13:105  OLD_TOTAL_NG %
% Rung: 6 %
SOR MOV L13:36 L13:92 EOR
%   L13:36  ONES %
%   L13:92  OLD_ONES %
% Rung: 7 %
SOR END EOR

LADDER 246 "SPEED BOT"    % high speed %
